// TIA Portal V18 export
TYPE "PartStatus_Enum"
   STRUCT
      PS_0_NO_PART : Int := 0;   // Empty / No part (Reset state)
      PS_100_GRIPPED_OK : Int := 100;   // Part ready for process / Gripped by robot (Grip OK)
      PS_110_OK_PART : Int := 110;   // OK part (Standard confirmation after scan or operation)
      PS_150_NG_GENERAL_ERROR : Int := 150;   // NG part (General scan or presence error)
      PS_151_NG_BARCODE_MISMATCH : Int := 151;   // NG â€“ Barcode Error (Mismatch)
      PS_152_NG_CODE_NO_READ : Int := 152;   // NG â€“ Code reading unsuccessful (No Read)
      PS_155_NG_ROBOT_SPECIFIC_ERROR : Int := 155;   // NG â€“ Specific error from Robot 2
      PS_180_ROTARY_SCAN_SPECIAL : Int := 180;   // Specific state for Rotary Shaft Scan (A1)
      PS_199_OPERATION_COMPLETED : Int := 199;   // Operation completed (Waiting for release/transfer)
      PS_220_PRESS1_INSERTED : Int := 220;   // Part inserted into press B1
      PS_250_PRESS1_IN_PROGRESS : Int := 250;   // Pressing B1 â€“ Start / In progress
      PS_251_PRESS1_NG_ERROR : Int := 251;   // Pressing B1 â€“ NG (Force/stroke error)
      PS_252_PRESS1_INTERRUPTED : Int := 252;   // Pressing B1 â€“ Interrupted
      PS_255_PRESS1_OK : Int := 255;   // Pressing B1 â€“ OK (Not yet finally released)
      PS_280_PRESS1_WAIT_REMOVE : Int := 280;   // Pressing B1 â€“ Waiting for removal
      PS_299_PRESS1_COMPLETED : Int := 299;   // Pressing B1 â€“ Completely finished
      PS_300_GLUING_START : Int := 300;   // Gluing â€“ Start / Preparation
      PS_310_GLUING_IN_PROGRESS : Int := 310;   // Glue application â€“ In progress
      PS_320_GLUE_INSP_IN_PROGRESS : Int := 320;   // Glue inspection (Vision) â€“ In progress
      PS_330_GLUE_INSP_NG : Int := 330;   // Glue inspection â€“ NG
      PS_351_GLUING_INTERM_POS1 : Int := 351;   // Gluing â€“ Intermediate state (Position 1)
      PS_352_GLUING_INTERM_POS2 : Int := 352;   // Gluing â€“ Intermediate state (Position 2)
      PS_358_GLUING_WAIT_ROBOT_HS : Int := 358;   // Gluing â€“ Waiting for robot handshake
      PS_359_GLUING_WAIT_ROBOT_HS2 : Int := 359;   // Gluing â€“ Waiting for robot handshake
      PS_380_GLUING_CRITICAL_ERROR : Int := 380;   // Gluing â€“ Critical device error
      PS_399_GLUING_COMPLETED : Int := 399;   // Gluing â€“ Completely finished (OK)
      PS_420_PRESS2_INSERTED : Int := 420;   // Part inserted into press B2
      PS_450_PRESS2_IN_PROGRESS : Int := 450;   // Pressing B2 â€“ Start / In progress
      PS_451_PRESS2_NG_ERROR : Int := 451;   // Pressing B2 â€“ NG (Force/stroke error)
      PS_452_PRESS2_INTERRUPTED : Int := 452;   // Pressing B2 â€“ Interrupted
      PS_455_PRESS2_OK : Int := 455;   // Pressing B2 â€“ OK
      PS_480_PRESS2_WAIT_REMOVE : Int := 480;   // Pressing B2 â€“ Waiting for removal
      PS_499_PRESS2_COMPLETED : Int := 499;   // Pressing B2 â€“ Completely finished
   END_STRUCT;
END_TYPE
